// TIA Portal project "EC PP Basik" (V17)

(* hardware
DEVICE "S7-1500/ET200MP station_2"  S7-1500 station
   slot 0: "Rail_0"  Rack  6ES7 590-1***0-0AA0
   slot 1: "PLC_1"  CPU 1511-1 PN  6ES7 511-1AK02-0AB0  V2.9
      slot 3: "CPU display_1"  6ES7591-1AA00-0AA0
      slot 32768: "PROFINET interface_1"  X1
         slot 32769: "Port_1"  X1 P1
         slot 32770: "Port_2"  X1 P2
      slot 34817: "Virtual CP interface port_1"  Virtual CP interface port  Virtual CP interface port
   slot 2: "DI 16x24VDC BA_1"  DI 16x24VDC BA  6ES7 521-1BH10-0AA0  V1.1
   slot 3: "DQ 16x24VDC/0.5A BA_1"  DQ 16x24VDC/0.5A BA  6ES7 522-1BH10-0AA0  V1.1
   slot 4: "AI 4xU/I/RTD/TC ST_1"  AI 4xU/I/RTD/TC ST  6ES7 531-7QD00-0AB0  V1.0
   slot 5: "AQ 4xU/I ST_1"  AQ 4xU/I ST  6ES7 532-5HD00-0AB0  V2.2
DEVICE "HMI_1"  KTP700 Basic PN
   slot 0: "HMI_1"  KTP700 Basic PN  6AV2 123-2GB03-0AX0  17.0.0.0
   slot 1: "HMI_RT_1"  KTP700 Basic PN  6AV2 123-2GB03-0AX0  17.0.0.0
   slot 5: "HMI_1.IE_CP_1"  PROFINET Interface  17.0.0.0
      slot 1: "PROFINET Interface_1"  PROFINET Interface
         slot 1: "Port_1"  Port
*)

// ===== PLC "PLC_1"  CPU 1511-1 PN =====

VAR_GLOBAL   // PLC tag table "IO"
   "Item at entry" AT %I0.0 : Bool;
   "Item at exit" AT %I0.1 : Bool;
   "Moving X" AT %I0.2 : Bool;
   "Moving Z" AT %I0.3 : Bool;
   "Item detected" AT %I0.4 : Bool;
   "Start" AT %I0.5 : Bool;
   "Reset" AT %I0.6 : Bool;
   "Stop" AT %I0.7 : Bool;
   "Emergency stop" AT %I1.0 : Bool;
   "Auto" AT %I1.1 : Bool;
   "FACTORY I/O (Running)" AT %I1.2 : Bool;
   "Manual" AT %I1.3 : Bool;
   "Entry conveyor" AT %Q0.0 : Bool;
   "Exit conveyor" AT %Q0.1 : Bool;
   "Move X" AT %Q0.2 : Bool;
   "Move Z" AT %Q0.3 : Bool;
   "Grab" AT %Q0.4 : Bool;
   "Start light" AT %Q0.5 : Bool;
   "Reset light" AT %Q0.6 : Bool;
   "Stop light" AT %Q0.7 : Bool;
   "Emitter" AT %Q1.0 : Bool;
   "Remover" AT %Q1.1 : Bool;
   "Counter" AT %QW30 : Int;
END_VAR

DATA_BLOCK "HMI_data"   // DB2
{ S7_Optimized_Access := 'TRUE' }
VERSION : 0.1
   VAR
      Start : Bool;
      Stop : Bool;
      Reset : Bool;
      Flanker : Struct
         Flank1 : Bool;
         Flank2 : Bool;
         Flank3 : Bool;
         Flank4 : Bool;
         Flank5 : Bool;
         Flank6 : Bool;
         Flank7 : Bool;
         Flank8 : Bool;
         Flank9 : Bool;
         Flank10 : Bool;
         Flank11 : Bool;
         Flank12 : Bool;
         Flank13 : Bool;
         Flank14 : Bool;
         Flank15 : Bool;
         Flank16 : Bool;
         Flank17 : Bool;
         Flank18 : Bool;
         Flank19 : Bool;
         Flank20 : Bool;
         Flank21 : Bool;
         Flank22 : Bool;
         Flank23 : Bool;
         Flank24 : Bool;
         Flank25 : Bool;
      END_STRUCT;
      Sekavensord : Int;
   END_VAR
BEGIN
END_DATA_BLOCK

// folder: System blocks/Program resources

DATA_BLOCK "IEC_Timer_0_DB"   // DB1
{ S7_Optimized_Access := 'TRUE' }
AUTHOR : Simatic
FAMILY : IEC
NAME : IEC_TMR
VERSION : 1.0
// stored: InstanceOfName IEC_TIMER
"IEC_TIMER"
BEGIN
END_DATA_BLOCK

DATA_BLOCK "IEC_Timer_0_DB_1"   // DB3
{ S7_Optimized_Access := 'TRUE' }
AUTHOR : Simatic
FAMILY : IEC
NAME : IEC_TMR
VERSION : 1.0
// stored: InstanceOfName IEC_TIMER
"IEC_TIMER"
BEGIN
END_DATA_BLOCK

// folder: (top level)

FUNCTION "HMI" : Void   // FC1, LAD
{ S7_Optimized_Access := 'TRUE' }
VERSION : 0.1
   VAR_TEMP   // added for the SCL form of the ladder/FBD networks
      _w1 : Bool;
   END_VAR
BEGIN

REGION Network 1: Starta sekvensen
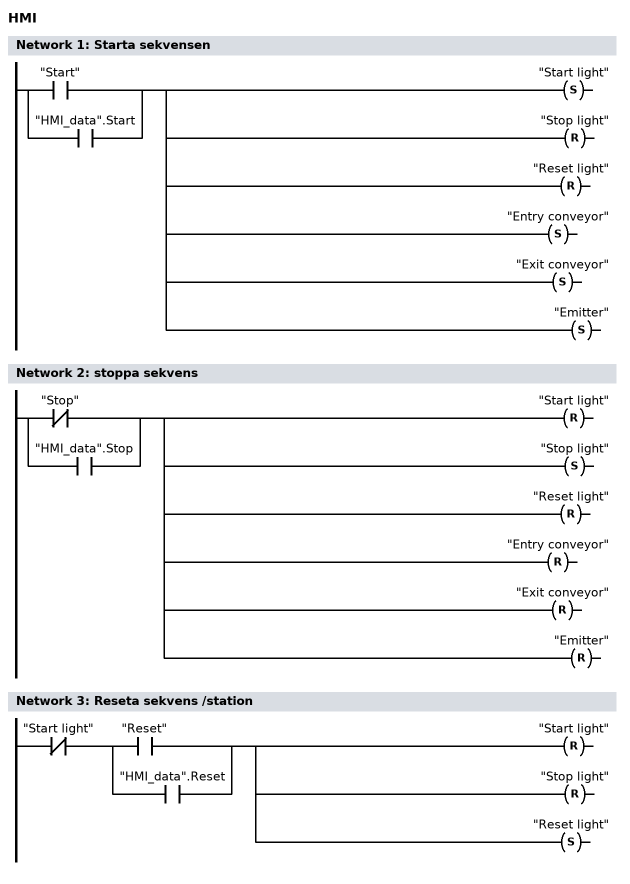
   RUNG wire#powerrail
      Contact( "Start" )
      wire#w1
      S_Coil( "Start light" )
   END_RUNG
   RUNG wire#powerrail
      Contact( "HMI_data".Start )
   END_RUNG wire#w1
   RUNG wire#w1
      R_Coil( "Stop light" )
   END_RUNG
   RUNG wire#w1
      R_Coil( "Reset light" )
   END_RUNG
   RUNG wire#w1
      S_Coil( "Entry conveyor" )
   END_RUNG
   RUNG wire#w1
      S_Coil( "Exit conveyor" )
   END_RUNG
   RUNG wire#w1
      S_Coil( "Emitter" )
   END_RUNG
   // the same network as SCL:
   IF "Start" OR "HMI_data".Start THEN
       "Start light" := TRUE;
       "Stop light" := FALSE;
       "Reset light" := FALSE;
       "Entry conveyor" := TRUE;
       "Exit conveyor" := TRUE;
       "Emitter" := TRUE;
   END_IF;
END_REGION

REGION Network 2: stoppa sekvens
   RUNG wire#powerrail
      I_Contact( "Stop" )
      wire#w1
      R_Coil( "Start light" )
   END_RUNG
   RUNG wire#powerrail
      Contact( "HMI_data".Stop )
   END_RUNG wire#w1
   RUNG wire#w1
      S_Coil( "Stop light" )
   END_RUNG
   RUNG wire#w1
      R_Coil( "Reset light" )
   END_RUNG
   RUNG wire#w1
      R_Coil( "Entry conveyor" )
   END_RUNG
   RUNG wire#w1
      R_Coil( "Exit conveyor" )
   END_RUNG
   RUNG wire#w1
      R_Coil( "Emitter" )
   END_RUNG
   // the same network as SCL:
   IF NOT "Stop" OR "HMI_data".Stop THEN
       "Start light" := FALSE;
       "Stop light" := TRUE;
       "Reset light" := FALSE;
       "Entry conveyor" := FALSE;
       "Exit conveyor" := FALSE;
       "Emitter" := FALSE;
   END_IF;
END_REGION

REGION Network 3: Reseta sekvens /station
   RUNG wire#powerrail
      I_Contact( "Start light" )
      wire#w1
      Contact( "Reset" )
      wire#w2
      R_Coil( "Start light" )
   END_RUNG
   RUNG wire#w1
      Contact( "HMI_data".Reset )
   END_RUNG wire#w2
   RUNG wire#w2
      R_Coil( "Stop light" )
   END_RUNG
   RUNG wire#w2
      S_Coil( "Reset light" )
   END_RUNG
   // the same network as SCL:
   #_w1 := NOT "Start light" AND ("Reset" OR "HMI_data".Reset);
   IF #_w1 THEN
       "Start light" := FALSE;
       "Stop light" := FALSE;
       "Reset light" := TRUE;
   END_IF;
END_REGION
END_FUNCTION

FUNCTION "Hmi_1" : Void   // FC2, LAD
{ S7_Optimized_Access := 'TRUE' }
VERSION : 0.1
   VAR_INPUT
      Start : Bool;
      Stop : Bool;
      Reset : Bool;
   END_VAR
   VAR_IN_OUT
      "Start light" : Bool;
      "Stop light" : Bool;
      "Reset light" : Bool;
   END_VAR
   VAR_TEMP   // added for the SCL form of the ladder/FBD networks
      _w1 : Bool;
   END_VAR
BEGIN

REGION Network 1: start logik
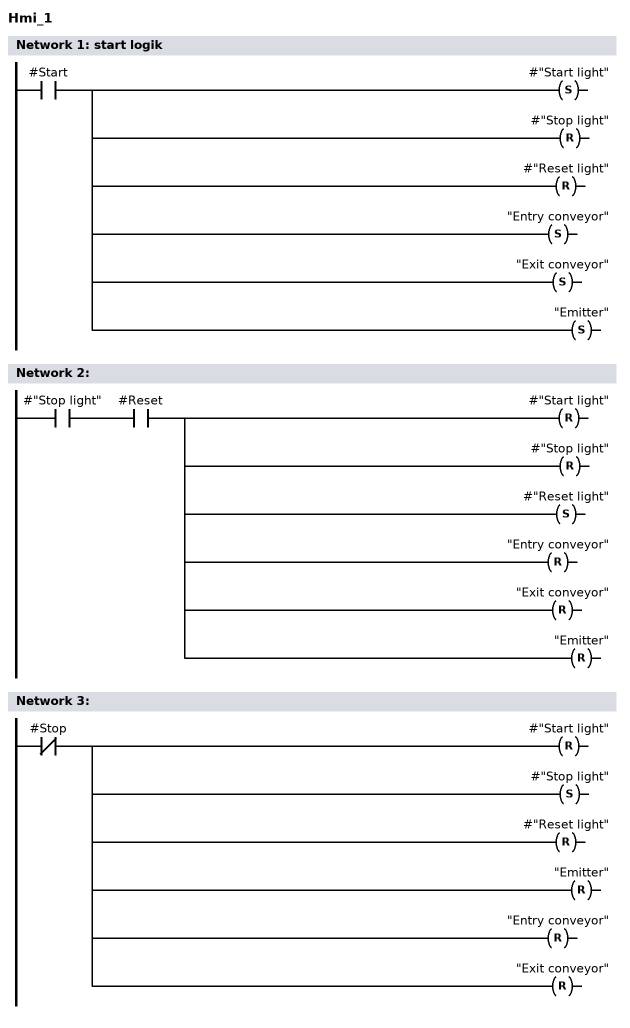
   RUNG wire#powerrail
      Contact( #Start )
      wire#w1
      S_Coil( #"Start light" )
   END_RUNG
   RUNG wire#w1
      R_Coil( #"Stop light" )
   END_RUNG
   RUNG wire#w1
      R_Coil( #"Reset light" )
   END_RUNG
   RUNG wire#w1
      S_Coil( "Entry conveyor" )
   END_RUNG
   RUNG wire#w1
      S_Coil( "Exit conveyor" )
   END_RUNG
   RUNG wire#w1
      S_Coil( "Emitter" )
   END_RUNG
   // the same network as SCL:
   IF #Start THEN
       #"Start light" := TRUE;
       #"Stop light" := FALSE;
       #"Reset light" := FALSE;
       "Entry conveyor" := TRUE;
       "Exit conveyor" := TRUE;
       "Emitter" := TRUE;
   END_IF;
END_REGION

REGION Network 2
   RUNG wire#powerrail
      Contact( #"Stop light" )
      Contact( #Reset )
      wire#w1
      R_Coil( #"Start light" )
   END_RUNG
   RUNG wire#w1
      R_Coil( #"Stop light" )
   END_RUNG
   RUNG wire#w1
      S_Coil( #"Reset light" )
   END_RUNG
   RUNG wire#w1
      R_Coil( "Entry conveyor" )
   END_RUNG
   RUNG wire#w1
      R_Coil( "Exit conveyor" )
   END_RUNG
   RUNG wire#w1
      R_Coil( "Emitter" )
   END_RUNG
   // the same network as SCL:
   IF #"Stop light" AND #Reset THEN #"Start light" := FALSE; END_IF;
   #_w1 := #"Stop light" AND #Reset;
   IF #_w1 THEN
       #"Stop light" := FALSE;
       #"Reset light" := TRUE;
       "Entry conveyor" := FALSE;
       "Exit conveyor" := FALSE;
       "Emitter" := FALSE;
   END_IF;
END_REGION

REGION Network 3
   RUNG wire#powerrail
      I_Contact( #Stop )
      wire#w1
      R_Coil( #"Start light" )
   END_RUNG
   RUNG wire#w1
      S_Coil( #"Stop light" )
   END_RUNG
   RUNG wire#w1
      R_Coil( #"Reset light" )
   END_RUNG
   RUNG wire#w1
      R_Coil( "Emitter" )
   END_RUNG
   RUNG wire#w1
      R_Coil( "Entry conveyor" )
   END_RUNG
   RUNG wire#w1
      R_Coil( "Exit conveyor" )
   END_RUNG
   // the same network as SCL:
   IF NOT #Stop THEN
       #"Start light" := FALSE;
       #"Stop light" := TRUE;
       #"Reset light" := FALSE;
       "Emitter" := FALSE;
       "Entry conveyor" := FALSE;
       "Exit conveyor" := FALSE;
   END_IF;
END_REGION
END_FUNCTION

FUNCTION "PP sekvens" : Void   // FC3, LAD
{ S7_Optimized_Access := 'TRUE' }
VERSION : 0.1
   VAR_TEMP   // added for the SCL form of the ladder/FBD networks
      _w1 : Bool;
      _w2 : Bool;
   END_VAR
BEGIN

REGION Network 1: sek0 resetar conveyors väntar på item at entry
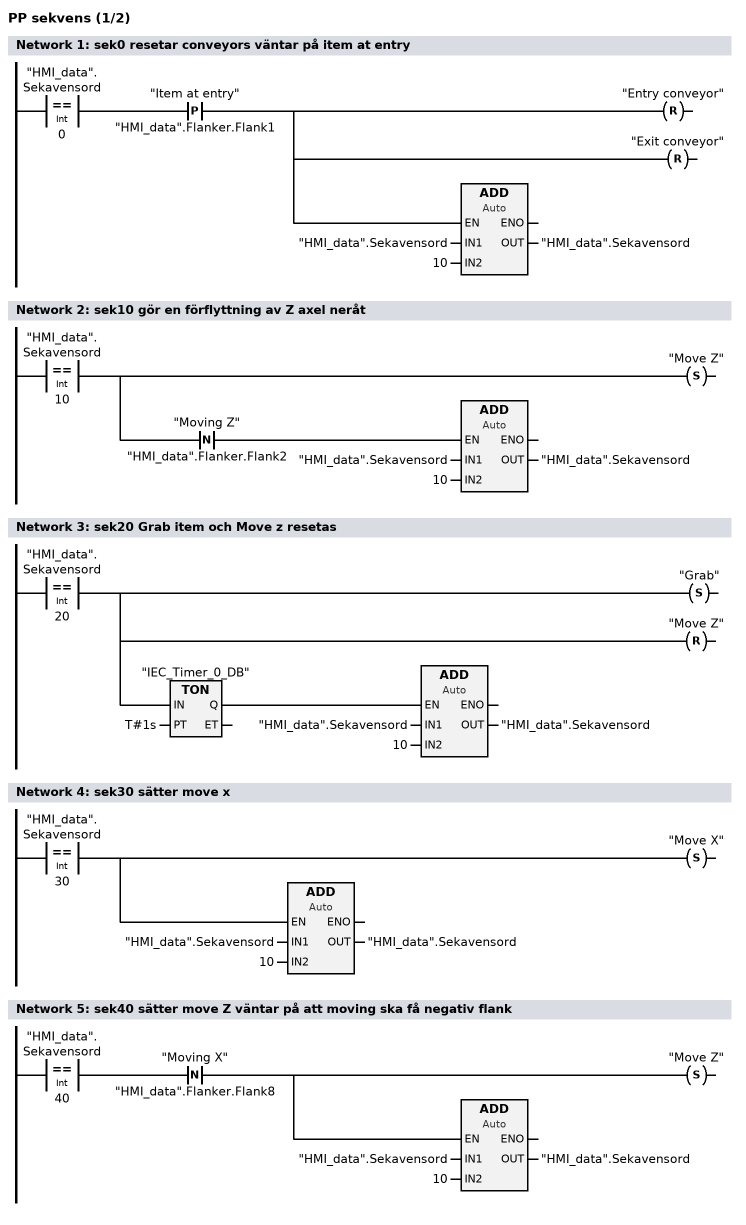
   RUNG wire#powerrail
      { S7_Templates := "SrcType := Int" } EQ_Contact(in1 := "HMI_data".Sekavensord, in2 := 0)
      P_Contact(operand := "Item at entry", bit := "HMI_data".Flanker.Flank1)
      wire#w1
      R_Coil( "Entry conveyor" )
   END_RUNG
   RUNG wire#w1
      R_Coil( "Exit conveyor" )
   END_RUNG
   RUNG wire#w1
      Add(in1 := "HMI_data".Sekavensord, in2 := 10, out => "HMI_data".Sekavensord)
   END_RUNG
   // the same network as SCL:
   #_w1 := ("HMI_data".Sekavensord = 0) AND "Item at entry" AND NOT "HMI_data".Flanker.Flank1;   // rising edge of "Item at entry"
   "HMI_data".Flanker.Flank1 := "Item at entry";
   IF #_w1 THEN
       "Entry conveyor" := FALSE;
       "Exit conveyor" := FALSE;
       "HMI_data".Sekavensord := "HMI_data".Sekavensord + 10;
   END_IF;
END_REGION

REGION Network 2: sek10 gör en förflyttning av Z axel neråt
   RUNG wire#powerrail
      { S7_Templates := "SrcType := Int" } EQ_Contact(in1 := "HMI_data".Sekavensord, in2 := 10)
      wire#w1
      S_Coil( "Move Z" )
   END_RUNG
   RUNG wire#w1
      N_Contact(operand := "Moving Z", bit := "HMI_data".Flanker.Flank2)
      Add(in1 := "HMI_data".Sekavensord, in2 := 10, out => "HMI_data".Sekavensord)
   END_RUNG
   // the same network as SCL:
   #_w1 := "HMI_data".Sekavensord = 10;
   IF #_w1 THEN "Move Z" := TRUE; END_IF;
   #_w2 := #_w1 AND NOT "Moving Z" AND "HMI_data".Flanker.Flank2;   // falling edge of "Moving Z"
   "HMI_data".Flanker.Flank2 := "Moving Z";
   IF #_w2 THEN "HMI_data".Sekavensord := "HMI_data".Sekavensord + 10; END_IF;
END_REGION

REGION Network 3: sek20 Grab item och Move z resetas
   #_w1 := "HMI_data".Sekavensord = 20;
   IF #_w1 THEN
       "Grab" := TRUE;
       "Move Z" := FALSE;
   END_IF;
   "IEC_Timer_0_DB".TON(IN := #_w1, PT := T#1s);
   IF "IEC_Timer_0_DB".Q THEN "HMI_data".Sekavensord := "HMI_data".Sekavensord + 10; END_IF;
END_REGION

REGION Network 4: sek30 sätter move x
   RUNG wire#powerrail
      { S7_Templates := "SrcType := Int" } EQ_Contact(in1 := "HMI_data".Sekavensord, in2 := 30)
      wire#w1
      S_Coil( "Move X" )
   END_RUNG
   RUNG wire#w1
      Add(in1 := "HMI_data".Sekavensord, in2 := 10, out => "HMI_data".Sekavensord)
   END_RUNG
   // the same network as SCL:
   IF "HMI_data".Sekavensord = 30 THEN
       "Move X" := TRUE;
       "HMI_data".Sekavensord := "HMI_data".Sekavensord + 10;
   END_IF;
END_REGION

REGION Network 5: sek40 sätter move Z väntar på att moving ska få negativ flank
   RUNG wire#powerrail
      { S7_Templates := "SrcType := Int" } EQ_Contact(in1 := "HMI_data".Sekavensord, in2 := 40)
      N_Contact(operand := "Moving X", bit := "HMI_data".Flanker.Flank8)
      wire#w1
      S_Coil( "Move Z" )
   END_RUNG
   RUNG wire#w1
      Add(in1 := "HMI_data".Sekavensord, in2 := 10, out => "HMI_data".Sekavensord)
   END_RUNG
   // the same network as SCL:
   #_w1 := ("HMI_data".Sekavensord = 40) AND NOT "Moving X" AND "HMI_data".Flanker.Flank8;   // falling edge of "Moving X"
   "HMI_data".Flanker.Flank8 := "Moving X";
   IF #_w1 THEN
       "Move Z" := TRUE;
       "HMI_data".Sekavensord := "HMI_data".Sekavensord + 10;
   END_IF;
END_REGION

REGION Network 6: sek50 reset Grab släpper detalj på exit conveyor
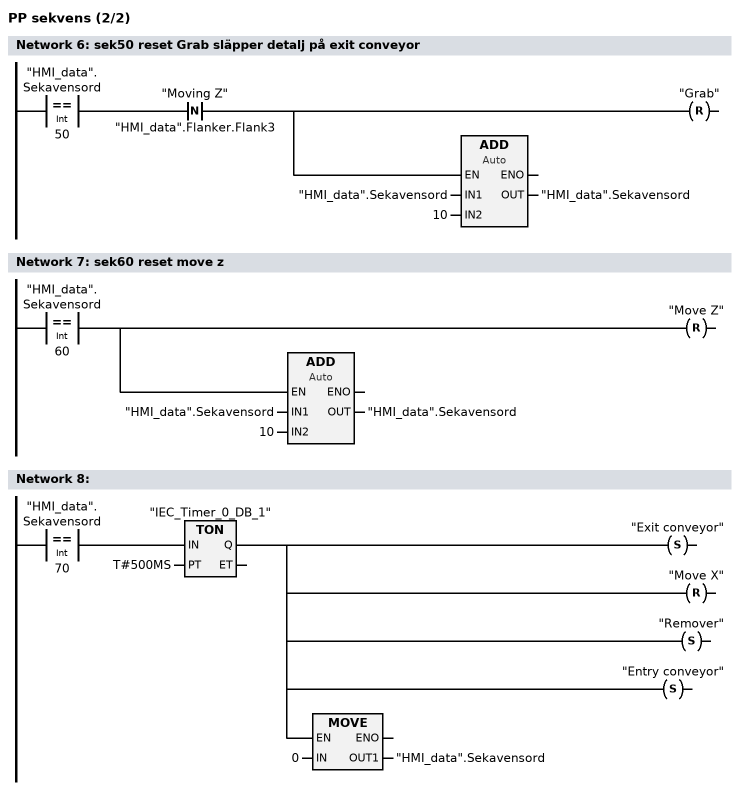
   RUNG wire#powerrail
      { S7_Templates := "SrcType := Int" } EQ_Contact(in1 := "HMI_data".Sekavensord, in2 := 50)
      N_Contact(operand := "Moving Z", bit := "HMI_data".Flanker.Flank3)
      wire#w1
      R_Coil( "Grab" )
   END_RUNG
   RUNG wire#w1
      Add(in1 := "HMI_data".Sekavensord, in2 := 10, out => "HMI_data".Sekavensord)
   END_RUNG
   // the same network as SCL:
   #_w1 := ("HMI_data".Sekavensord = 50) AND NOT "Moving Z" AND "HMI_data".Flanker.Flank3;   // falling edge of "Moving Z"
   "HMI_data".Flanker.Flank3 := "Moving Z";
   IF #_w1 THEN
       "Grab" := FALSE;
       "HMI_data".Sekavensord := "HMI_data".Sekavensord + 10;
   END_IF;
END_REGION

REGION Network 7: sek60 reset move z
   RUNG wire#powerrail
      { S7_Templates := "SrcType := Int" } EQ_Contact(in1 := "HMI_data".Sekavensord, in2 := 60)
      wire#w1
      R_Coil( "Move Z" )
   END_RUNG
   RUNG wire#w1
      Add(in1 := "HMI_data".Sekavensord, in2 := 10, out => "HMI_data".Sekavensord)
   END_RUNG
   // the same network as SCL:
   IF "HMI_data".Sekavensord = 60 THEN
       "Move Z" := FALSE;
       "HMI_data".Sekavensord := "HMI_data".Sekavensord + 10;
   END_IF;
END_REGION

REGION Network 8
   "IEC_Timer_0_DB_1".TON(IN := "HMI_data".Sekavensord = 70, PT := T#500MS);
   IF "IEC_Timer_0_DB_1".Q THEN
       "Exit conveyor" := TRUE;
       "Move X" := FALSE;
       "Remover" := TRUE;
       "Entry conveyor" := TRUE;
       "HMI_data".Sekavensord := 0;
   END_IF;
END_REGION
END_FUNCTION

FUNCTION "Raknare" : Void   // FC4, LAD
{ S7_Optimized_Access := 'TRUE' }
VERSION : 0.1
   VAR_TEMP   // added for the SCL form of the ladder/FBD networks
      _w1 : Bool;
   END_VAR
BEGIN

REGION Network 1
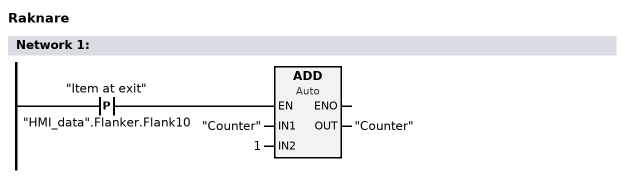
   RUNG wire#powerrail
      P_Contact(operand := "Item at exit", bit := "HMI_data".Flanker.Flank10)
      Add(in1 := "Counter", in2 := 1, out => "Counter")
   END_RUNG
   // the same network as SCL:
   #_w1 := "Item at exit" AND NOT "HMI_data".Flanker.Flank10;   // rising edge of "Item at exit"
   "HMI_data".Flanker.Flank10 := "Item at exit";
   IF #_w1 THEN "Counter" := "Counter" + 1; END_IF;
END_REGION
END_FUNCTION

ORGANIZATION_BLOCK "Main"   // OB1, LAD, ProgramCycle
TITLE = "Main Program Sweep (Cycle)"
{ S7_Optimized_Access := 'TRUE' }
VERSION : 0.1
   VAR_INPUT
      Initial_Call : Bool;   // Initial call of this OB
      Remanence : Bool;   // =True, if remanent data are available
   END_VAR
BEGIN

REGION Network 1
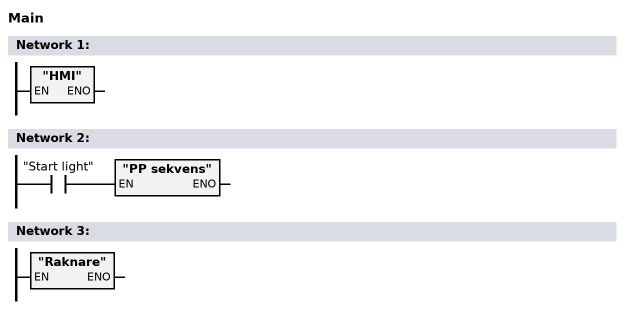
   RUNG wire#powerrail
      "HMI"()
   END_RUNG
   // the same network as SCL:
   "HMI"();
END_REGION

REGION Network 2
   RUNG wire#powerrail
      Contact( "Start light" )
      "PP sekvens"()
   END_RUNG
   // the same network as SCL:
   IF "Start light" THEN "PP sekvens"(); END_IF;
END_REGION

REGION Network 3
   RUNG wire#powerrail
      "Raknare"()
   END_RUNG
   // the same network as SCL:
   "Raknare"();
END_REGION
END_ORGANIZATION_BLOCK

(* ===== HMI "HMI_RT_1" =====
system functions are stored by id; their names below are inferred from use
connection "HMI_Connection_1": ETHERNET, SMART_S7_1500_OMS

HMI tags "Default tag table"
   "Tag_ScreenNumber" : UInt, internal
   "Start" : Bool = PLC Start AT %I0.5, 1 s
   "HMI_data_Start" : Bool = PLC HMI_data.Start, 1 s
   "HMI_data_Reset" : Bool = PLC HMI_data.Reset, 1 s
   "HMI_data_Stop" : Bool = PLC HMI_data.Stop, 1 s
   "Start light" : Bool = PLC "Start light" AT %Q0.5, 1 s
   "Stop light" : Bool = PLC "Stop light" AT %Q0.7, 1 s
   "Reset light" : Bool = PLC "Reset light" AT %Q0.6, 1 s
   "Counter" : Int = PLC Counter AT %QW30, 1 s

Template "Template_1" 800x480
   Button "Exit" at 714,429 size 71x50; TextOff 'Exit'; PictureOff "ExitRuntime_KTP700_Basic_PN_TR"; PictureOn "ExitRuntime_KTP700_Basic_PN_TR"
      on Release: StopRuntime(0)
   Button "Template_Button" at 614,429 size 71x50; TextOff 'Text'
   Button "Template_Button_1" at 514,429 size 71x50; TextOff 'Text'
   Button "Template_Button_2" at 414,429 size 71x50; TextOff 'Text'
   Button "Template_Button_3" at 314,429 size 71x50; TextOff 'Text'
   Button "Template_Button_4" at 214,429 size 71x50; TextOff 'Text'
   Button "Alarms" at 114,429 size 71x50; TextOff 'Alarms'; PictureOff "AlarmDisplay_KTP700_Basic_PN_TR"; PictureOn "AlarmDisplay_KTP700_Basic_PN_TR"
      on Release: function_ef3f5d25("Alarm window_Unacknowledged", -1)
   Button "Start screen" at 14,429 size 71x50; TextOff 'Start screen'; PictureOff "NavigateHome_KTP700_Basic_PN_TR"; PictureOn "NavigateHome_KTP700_Basic_PN_TR"
      on Release: ActivateScreen("Root screen", 0)
   SymbolicIOField "Symbolic_IO_Field_Screen" at 93,9 size 600x33; TextOff '0'; TextOn '1'; TextList "TextList_ScreenNames"
      ProcessValue <- "Tag_ScreenNumber"
      on Change: ActivateScreenByNumber("Tag_ScreenNumber", 0)
   DateTimeField "HmiScreenItemData" at 695,25 size 105x25
   DateTimeField "HmiScreenItemData_1" at 695,0 size 105x25
   GraphicView "Logo" at 0,0 size 91x51; Picture "Logo of HMI_1"

screen "Root screen" 800x480, template "Template_1"
   on GenerateScreen: SetTag("Tag_ScreenNumber", 1)
   Button "HmiScreenItemData" at 36,87 size 159x47; TextOff 'Start stop'; PictureOff "Navigates to Start stop for KTP700 Basic+ PN 17.0.0.0"; PictureOn "Navigates to Start stop for KTP700 Basic+ PN 17.0.0.0"
      on Release: ActivateScreen("Start stop", 0)
   Button "HmiScreenItemData_1" at 36,146 size 159x47; TextOff 'statestik'; PictureOff "Navigates to statestik for KTP700 Basic+ PN 17.0.0.0"; PictureOn "Navigates to statestik for KTP700 Basic+ PN 17.0.0.0"
      on Release: ActivateScreen("statestik", 0)
   Button "HmiScreenItemData_3" at 36,205 size 159x47; TextOff 'System screens'; PictureOff "Navigates to System screens for KTP700 Basic+ PN 17.0.0.0"; PictureOn "Navigates to System screens for KTP700 Basic+ PN 17.0.0.0"
      on Release: ActivateScreen("System screens", 0)

screen "Start stop" 800x480, template "Template_1"
   on GenerateScreen: SetTag("Tag_ScreenNumber", 2)
   TextField "HmiScreenItemData" at 92,57 size 640x25; Text 'Start stop'
   Button "Back" at 0,57 size 159x47; TextOff 'Tillbaka'; TextOn 'Back'
      on Release: ActivateScreen("Root screen", 0)
   Button "Button_1" at 92,217 size 124x32; TextOff 'Start Knapp'
      on Press: function_b14e0dd5("HMI_data_Start", 0)
      Appearance <- "Start light"
   Button "Button_2" at 249,217 size 124x32; TextOff 'Stop Knapp'
      on Press: function_b14e0dd5("HMI_data_Stop", 0)
      Appearance <- "Stop light"
   Button "Button_3" at 406,217 size 124x32; TextOff 'Reset Knapp'
      on Press: function_b14e0dd5("HMI_data_Reset", 0)
      Appearance <- "Reset light"
   IOField "I/O field_1" at 92,326 size 96x32; FormatPattern 9999
      ProcessValue <- "Counter"
   TextField "Text field_1" at 92,294 size 107x23; Text 'Totalt körda'

screen "statestik" 800x480, template "Template_1"
   on GenerateScreen: SetTag("Tag_ScreenNumber", 3)
   TextField "HmiScreenItemData" at 80,225 size 640x25; Text 'statestik'
   Button "Back" at 1,52 size 159x47; TextOff 'Back'
      on Release: ActivateScreen("Root screen", 0)

screen "System screens" 800x480, template "Template_1"
   on GenerateScreen: SetTag("Tag_ScreenNumber", 4)
   Button "Back" at 1,52 size 159x47; TextOff 'Back'
      on Release: ActivateScreen("Root screen", 0)
   Button "HmiScreenItemData" at 36,146 size 159x47; TextOff 'User administration'; PictureOff "Navigates to User administration for KTP700 Basic+ PN 17.0.0.0"; PictureOn "Navigates to User administration for KTP700 Basic+ PN 17.0.0.0"
      on Release: ActivateScreen("User administration", 0)
   Button "HmiScreenItemData_1" at 36,205 size 159x47; TextOff 'Different jobs'; PictureOff "Navigates to Different jobs for KTP700 Basic+ PN 17.0.0.0"; PictureOn "Navigates to Different jobs for KTP700 Basic+ PN 17.0.0.0"
      on Release: ActivateScreen("Different jobs", 0)

screen "User administration" 800x480, template "Template_1"
   on GenerateScreen: SetTag("Tag_ScreenNumber", 5)
   UserView "HmiScreenItemData" at 1,100 size 796x321
   Button "Back" at 1,52 size 159x47; TextOff 'Back'
      on Release: ActivateScreen("System screens", 0)

screen "Different jobs" 800x480, template "Template_1"
   on GenerateScreen: SetTag("Tag_ScreenNumber", 6)
   Button "Toggle language" at 36,146 size 159x47; TextOff 'Toggle language'
      on Release: function_fb9197e8(-1)
   Button "Back" at 1,52 size 159x47; TextOff 'Back'
      on Release: ActivateScreen("System screens", 0)
*)